// Mitsubishi GX Works2 project: THIET BI VE SINH STATOR   PLC: FX3S

PROGRAM MAIN
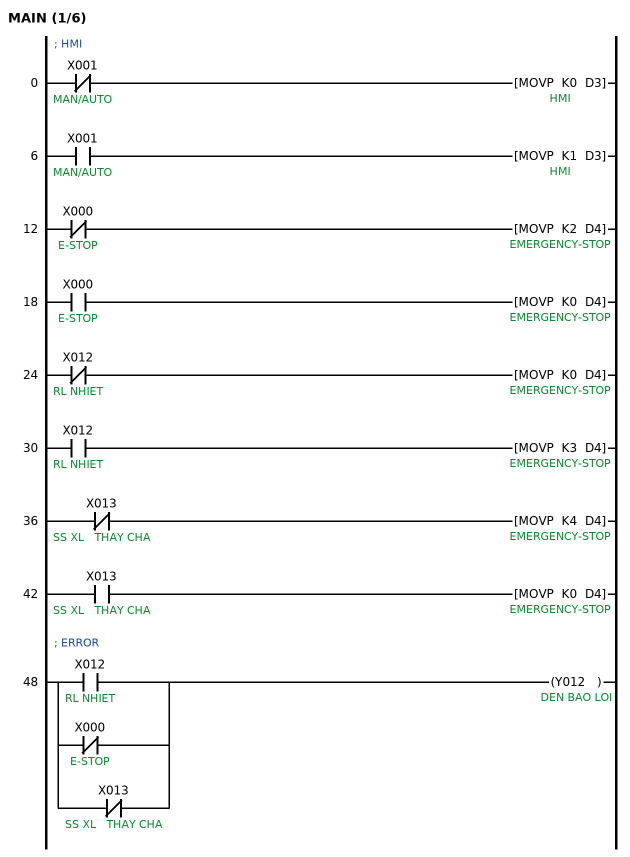
; HMI
0     LDI     X001  ; MAN/AUTO
      MOVP    K0 D3  ; HMI
6     LD      X001  ; MAN/AUTO
      MOVP    K1 D3
12    LDI     X000  ; E-STOP
      MOVP    K2 D4  ; EMERGENCY-STOP
18    LD      X000  ; E-STOP
      MOVP    K0 D4
24    LDI     X012  ; RL NHIET
      MOVP    K0 D4
30    LD      X012  ; RL NHIET
      MOVP    K3 D4
36    LDI     X013  ; SS XL   THAY CHA
      MOVP    K4 D4
42    LD      X013  ; SS XL   THAY CHA
      MOVP    K0 D4
; ERROR
48    LD      X012  ; RL NHIET
      ORI     X000  ; E-STOP
      ORI     X013  ; SS XL   THAY CHA
      OUT     Y012  ; DEN BAO LOI
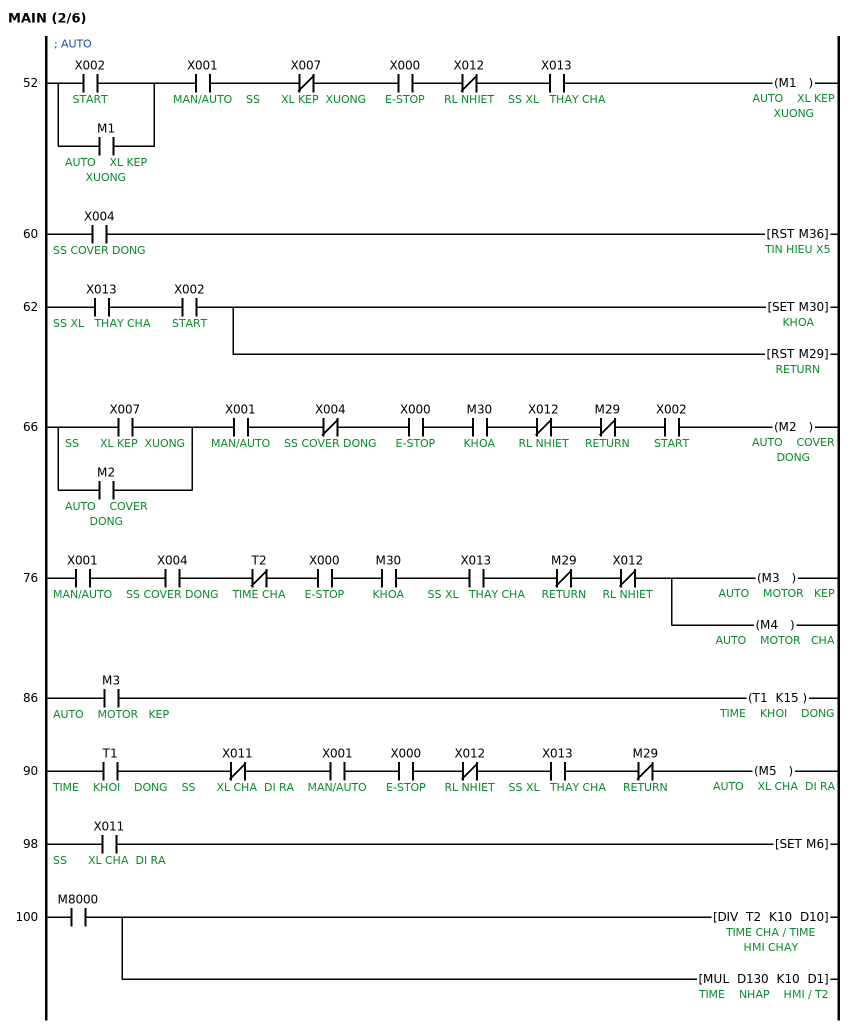
; AUTO
52    LD      X002  ; START
      OR      M1  ; AUTO    XL KEP  XUONG
      AND     X001  ; MAN/AUTO
      ANI     X007  ; SS      XL KEP  XUONG
      AND     X000  ; E-STOP
      ANI     X012  ; RL NHIET
      AND     X013  ; SS XL   THAY CHA
      OUT     M1  ; AUTO    XL KEP  XUONG
60    LD      X004  ; SS COVER DONG
      RST     M36  ; TIN HIEU X5
62    LD      X013  ; SS XL   THAY CHA
      AND     X002  ; START
      SET     M30  ; KHOA
      RST     M29  ; RETURN
66    LD      X007  ; SS      XL KEP  XUONG
      OR      M2  ; AUTO    COVER   DONG
      AND     X001  ; MAN/AUTO
      ANI     X004  ; SS COVER DONG
      AND     X000  ; E-STOP
      AND     M30  ; KHOA
      ANI     X012  ; RL NHIET
      ANI     M29  ; RETURN
      AND     X002  ; START
      OUT     M2  ; AUTO    COVER   DONG
76    LD      X001  ; MAN/AUTO
      AND     X004  ; SS COVER DONG
      ANI     T2  ; TIME CHA
      AND     X000  ; E-STOP
      AND     M30  ; KHOA
      AND     X013  ; SS XL   THAY CHA
      ANI     M29  ; RETURN
      ANI     X012  ; RL NHIET
      OUT     M3  ; AUTO    MOTOR   KEP
      OUT     M4  ; AUTO    MOTOR   CHA
86    LD      M3  ; AUTO    MOTOR   KEP
      OUT     T1 K15  ; TIME    KHOI    DONG
90    LD      T1  ; TIME    KHOI    DONG
      ANI     X011  ; SS      XL CHA  DI RA
      AND     X001  ; MAN/AUTO
      AND     X000  ; E-STOP
      ANI     X012  ; RL NHIET
      AND     X013  ; SS XL   THAY CHA
      ANI     M29  ; RETURN
      OUT     M5  ; AUTO    XL CHA  DI RA
98    LD      X011  ; SS      XL CHA  DI RA
      SET     M6
100   LD      M8000
      DIV     T2 K10 D10  ; TIME    HMI CHAY
      MUL     D130 K10 D1  ; TIME    NHAP    HMI / T2
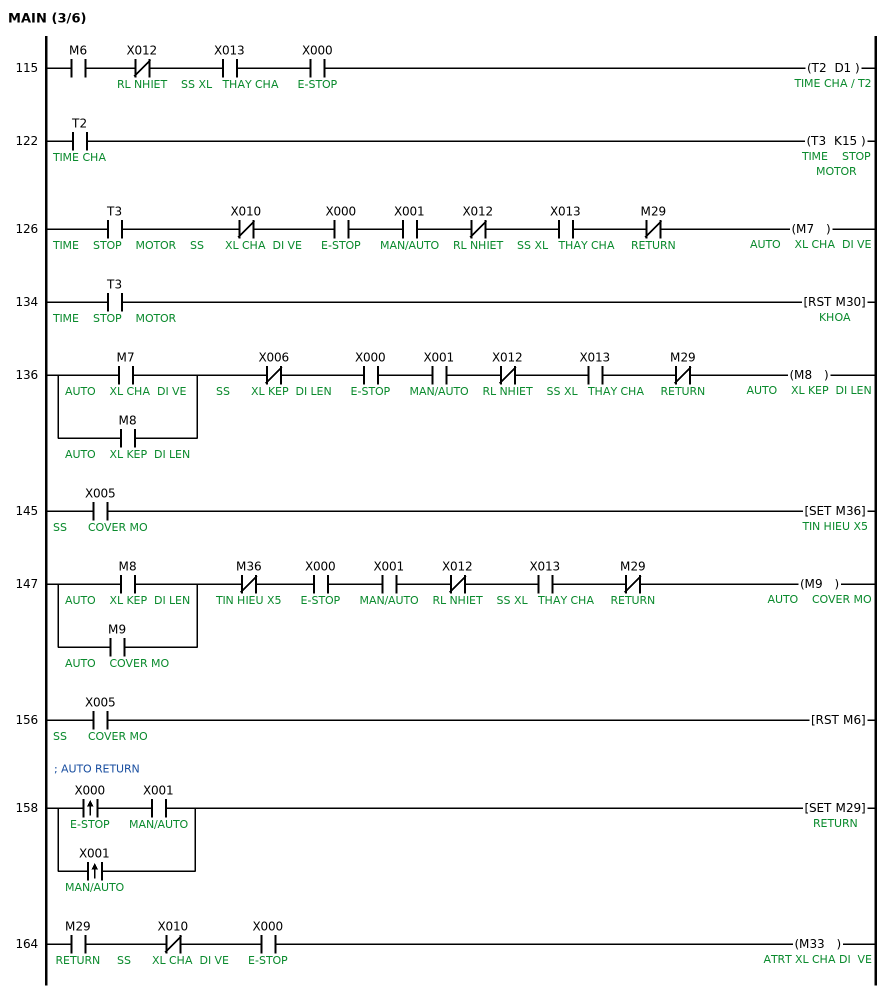
115   LD      M6
      ANI     X012  ; RL NHIET
      AND     X013  ; SS XL   THAY CHA
      AND     X000  ; E-STOP
      OUT     T2 D1  ; TIME CHA / T2
122   LD      T2  ; TIME CHA
      OUT     T3 K15  ; TIME    STOP    MOTOR
126   LD      T3  ; TIME    STOP    MOTOR
      ANI     X010  ; SS      XL CHA  DI VE
      AND     X000  ; E-STOP
      AND     X001  ; MAN/AUTO
      ANI     X012  ; RL NHIET
      AND     X013  ; SS XL   THAY CHA
      ANI     M29  ; RETURN
      OUT     M7  ; AUTO    XL CHA  DI VE
134   LD      T3  ; TIME    STOP    MOTOR
      RST     M30  ; KHOA
136   LD      M7  ; AUTO    XL CHA  DI VE
      OR      M8  ; AUTO    XL KEP  DI LEN
      ANI     X006  ; SS      XL KEP  DI LEN
      AND     X000  ; E-STOP
      AND     X001  ; MAN/AUTO
      ANI     X012  ; RL NHIET
      AND     X013  ; SS XL   THAY CHA
      ANI     M29  ; RETURN
      OUT     M8  ; AUTO    XL KEP  DI LEN
145   LD      X005  ; SS      COVER MO
      SET     M36  ; TIN HIEU X5
147   LD      M8  ; AUTO    XL KEP  DI LEN
      OR      M9  ; AUTO    COVER MO
      ANI     M36  ; TIN HIEU X5
      AND     X000  ; E-STOP
      AND     X001  ; MAN/AUTO
      ANI     X012  ; RL NHIET
      AND     X013  ; SS XL   THAY CHA
      ANI     M29  ; RETURN
      OUT     M9  ; AUTO    COVER MO
156   LD      X005  ; SS      COVER MO
      RST     M6
; AUTO RETURN
158   LDP     X000  ; E-STOP
      AND     X001  ; MAN/AUTO
      ORP     X001  ; MAN/AUTO
      SET     M29  ; RETURN
164   LD      M29  ; RETURN
      ANI     X010  ; SS      XL CHA  DI VE
      AND     X000  ; E-STOP
      OUT     M33  ; ATRT XL CHA DI  VE
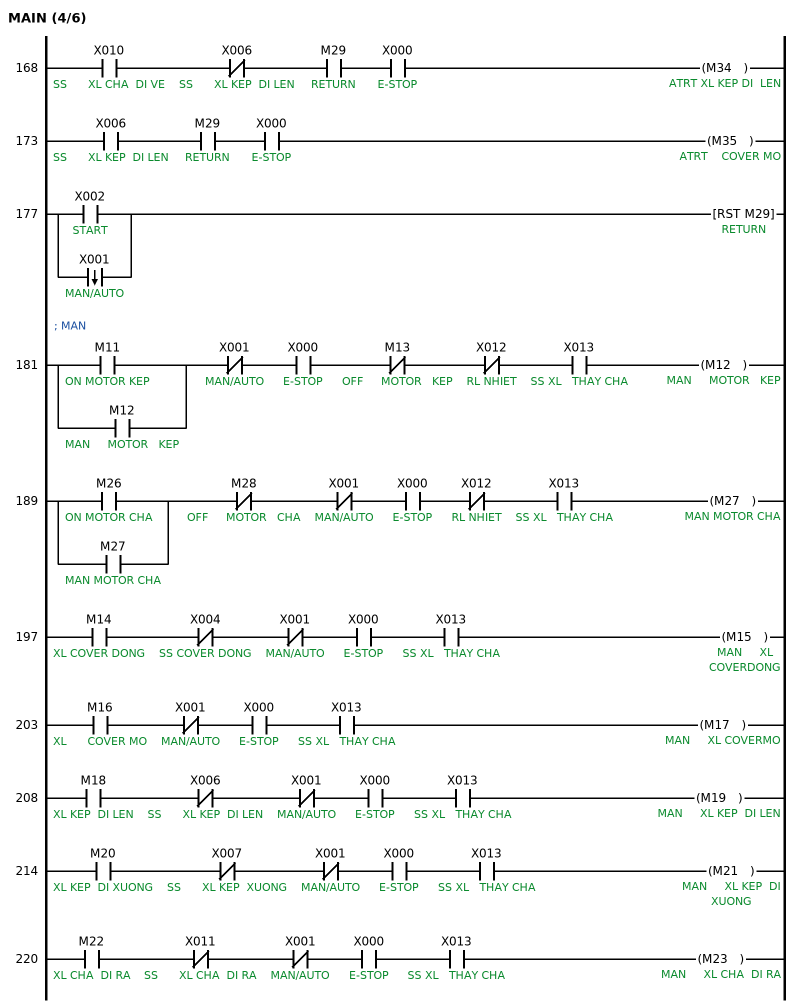
168   LD      X010  ; SS      XL CHA  DI VE
      ANI     X006  ; SS      XL KEP  DI LEN
      AND     M29  ; RETURN
      AND     X000  ; E-STOP
      OUT     M34  ; ATRT XL KEP DI  LEN
173   LD      X006  ; SS      XL KEP  DI LEN
      AND     M29  ; RETURN
      AND     X000  ; E-STOP
      OUT     M35  ; ATRT    COVER MO
177   LD      X002  ; START
      ORF     X001  ; MAN/AUTO
      RST     M29  ; RETURN
; MAN
181   LD      M11  ; ON MOTOR KEP
      OR      M12  ; MAN     MOTOR   KEP
      ANI     X001  ; MAN/AUTO
      AND     X000  ; E-STOP
      ANI     M13  ; OFF     MOTOR   KEP
      ANI     X012  ; RL NHIET
      AND     X013  ; SS XL   THAY CHA
      OUT     M12  ; MAN     MOTOR   KEP
189   LD      M26  ; ON MOTOR CHA
      OR      M27  ; MAN MOTOR CHA
      ANI     M28  ; OFF     MOTOR   CHA
      ANI     X001  ; MAN/AUTO
      AND     X000  ; E-STOP
      ANI     X012  ; RL NHIET
      AND     X013  ; SS XL   THAY CHA
      OUT     M27  ; MAN MOTOR CHA
197   LD      M14  ; XL COVER DONG
      ANI     X004  ; SS COVER DONG
      ANI     X001  ; MAN/AUTO
      AND     X000  ; E-STOP
      AND     X013  ; SS XL   THAY CHA
      OUT     M15  ; MAN     XL COVERDONG
203   LD      M16  ; XL      COVER MO
      ANI     X001  ; MAN/AUTO
      AND     X000  ; E-STOP
      AND     X013  ; SS XL   THAY CHA
      OUT     M17  ; MAN     XL COVERMO
208   LD      M18  ; XL KEP  DI LEN
      ANI     X006  ; SS      XL KEP  DI LEN
      ANI     X001  ; MAN/AUTO
      AND     X000  ; E-STOP
      AND     X013  ; SS XL   THAY CHA
      OUT     M19  ; MAN     XL KEP  DI LEN
214   LD      M20  ; XL KEP  DI XUONG
      ANI     X007  ; SS      XL KEP  XUONG
      ANI     X001  ; MAN/AUTO
      AND     X000  ; E-STOP
      AND     X013  ; SS XL   THAY CHA
      OUT     M21  ; MAN     XL KEP  DI XUONG
220   LD      M22  ; XL CHA  DI RA
      ANI     X011  ; SS      XL CHA  DI RA
      ANI     X001  ; MAN/AUTO
      AND     X000  ; E-STOP
      AND     X013  ; SS XL   THAY CHA
      OUT     M23  ; MAN     XL CHA  DI RA
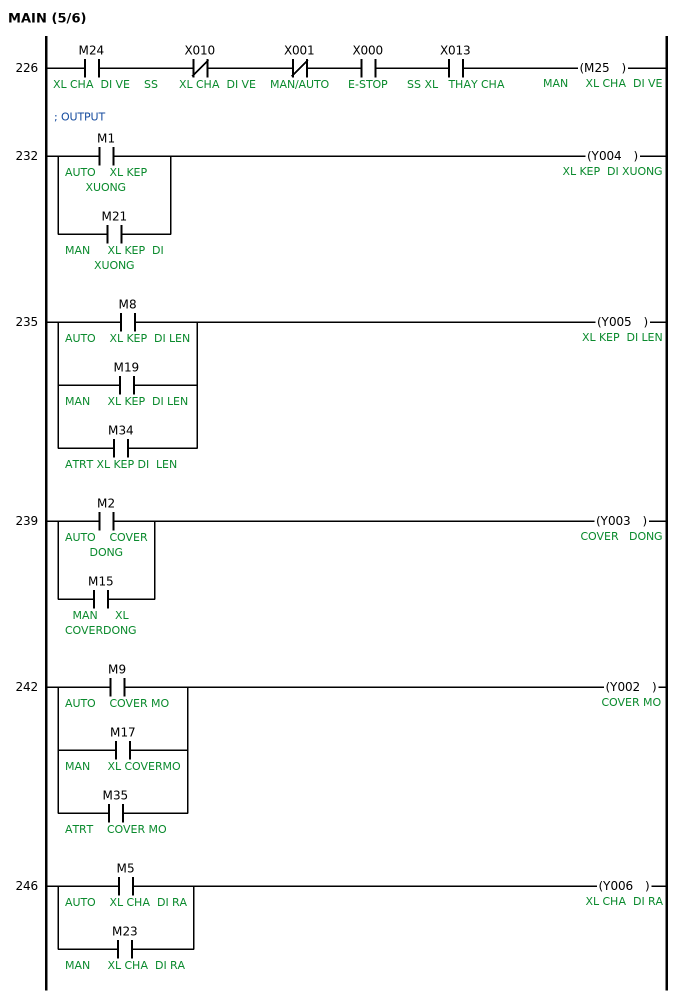
226   LD      M24  ; XL CHA  DI VE
      ANI     X010  ; SS      XL CHA  DI VE
      ANI     X001  ; MAN/AUTO
      AND     X000  ; E-STOP
      AND     X013  ; SS XL   THAY CHA
      OUT     M25  ; MAN     XL CHA  DI VE
; OUTPUT
232   LD      M1  ; AUTO    XL KEP  XUONG
      OR      M21  ; MAN     XL KEP  DI XUONG
      OUT     Y004  ; XL KEP  DI XUONG
235   LD      M8  ; AUTO    XL KEP  DI LEN
      OR      M19  ; MAN     XL KEP  DI LEN
      OR      M34  ; ATRT XL KEP DI  LEN
      OUT     Y005  ; XL KEP  DI LEN
239   LD      M2  ; AUTO    COVER   DONG
      OR      M15  ; MAN     XL COVERDONG
      OUT     Y003  ; COVER   DONG
242   LD      M9  ; AUTO    COVER MO
      OR      M17  ; MAN     XL COVERMO
      OR      M35  ; ATRT    COVER MO
      OUT     Y002  ; COVER MO
246   LD      M5  ; AUTO    XL CHA  DI RA
      OR      M23  ; MAN     XL CHA  DI RA
      OUT     Y006  ; XL CHA  DI RA
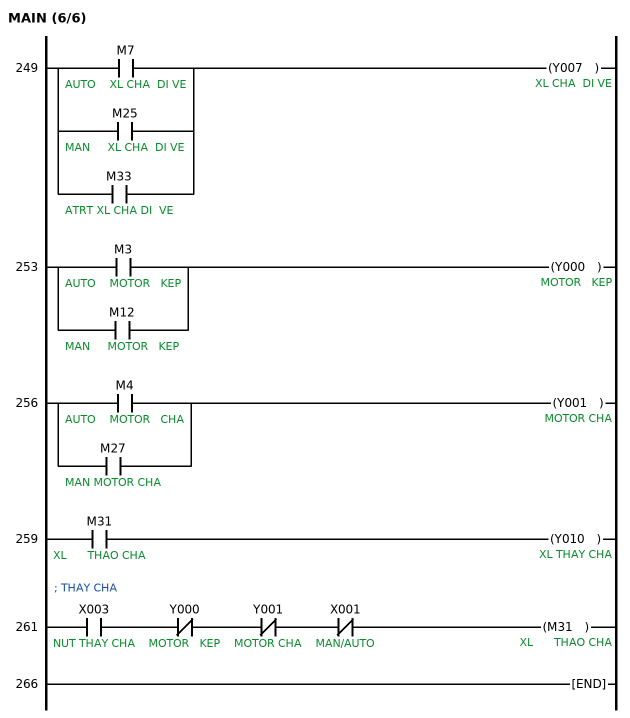
249   LD      M7  ; AUTO    XL CHA  DI VE
      OR      M25  ; MAN     XL CHA  DI VE
      OR      M33  ; ATRT XL CHA DI  VE
      OUT     Y007  ; XL CHA  DI VE
253   LD      M3  ; AUTO    MOTOR   KEP
      OR      M12  ; MAN     MOTOR   KEP
      OUT     Y000  ; MOTOR   KEP
256   LD      M4  ; AUTO    MOTOR   CHA
      OR      M27  ; MAN MOTOR CHA
      OUT     Y001  ; MOTOR CHA
259   LD      M31  ; XL      THAO CHA
      OUT     Y010  ; XL THAY CHA
; THAY CHA
261   LD      X003  ; NUT THAY CHA
      ANI     Y000  ; MOTOR   KEP
      ANI     Y001  ; MOTOR CHA
      ANI     X001  ; MAN/AUTO
      OUT     M31  ; XL      THAO CHA
266   END
END_PROGRAM

// device comments not shown above
Y011  ; DEN
M32  ; XL      THAO CHA DI VE
M37  ; TIN HIEU SS THAY CHA
T6  ; TIME    THAO CHA
D2  ; T3
D5  ; OVERLOAD
P1  ; AUTO
P2  ; MANUAL
P3  ; OUTPUT
P4  ; BAO LOI
P5  ; RETURN
